{attribute 'qualified_only'}
{attribute 'strict'}
TYPE eTcoDaqTests :
(
	Push := 10
);
END_TYPE

(* stored: Version 1.1.0.1
   DUT eTcoDaqTests: Id {26de48e7-e83b-0fca-07ab-ee65941e6af0} *)
